//==================================================================================================
//							Beckhoff Automation Poland
//									2.11.2018
//	Place to collect all module error, warning, ready etc flags. Here You can mute errors also.
// 
//	v1.0 	|| TC v 3.1.4022.25 		|| Pierwsza wersja
//==================================================================================================
PROGRAM P_ErrorCollection
VAR
	bOK										: BOOL;
	bWarning								: BOOL;
	bError									: BOOL;
	bFatalError								: BOOL;
END_VAR

bError := P_SystemDiagnostics.bError OR P_Template_SAFETY.bError; // And more....
// Collect flags - real
bWarning  								:= bWarning; 										// Collection
bError  								:= bError; 											// Collection
bFatalError  							:= bFatalError; 									// Collection
bOk										:= NOT (bWarning OR bError OR bFatalError);
// Pass to global, add mute if neccesary
GVL.bGeneralWarning  					:= bWarning;										// Pass
GVL.bGeneralError  						:= bError AND NOT GVL.bMuteGeneralError;			// Pass and mute
GVL.bGeneralFatalError  				:= bFatalError AND NOT GVL.bMuteGeneralFatalError;	// Pass and mute
GVL.bGeneralOK 							:= NOT GVL.bGeneralWarning OR GVL.bGeneralError OR GVL.bGeneralFatalError;
// Machine units ready flag
GVL.bAllUnitsReady 						:= NOT (P_Template.bError (*OR P_Template_CAM.bError*));	// All units
// After fatal error and auto mode machine reset is required
GVL.bRestartRequired					R= NOT GVL.bGeneralFatalError;
GVL.bRestartRequired					S= GVL.bGeneralFatalError AND (GVL_Machine.eMode = E_MachineMode.eAutomatic);

END_PROGRAM

(* stored: Version 1.1.0.1, ProductVersion 3.1.4022.12
   POU P_ErrorCollection: Id {12c6371e-2444-4a6d-b57d-58647b3301b7}, SpecialFunc None *)
